TYPE ST_PiezoStageCSP  EXTENDS ST_PiezoStage :
STRUCT
    (*CSP drive mode*)
    nFollowingError 		AT %I*: DINT;
END_STRUCT
END_TYPE

(* stored: Version 1.1.0.1
   DUT ST_PiezoStageCSP: Id {d2b946d8-0cf7-42b6-9e42-6c1a835d954a} *)
